PROGRAM PRG_HMI
VAR
	counter	: FB_Counter;
END_VAR

GVL_HMI.output_1:=  GVL_HMI.input_1 AND GVL_HMI.input_2;

counter(CTU:=GVL_HMI.btn_CTU ,
		CTD:=GVL_HMI.btn_CTD , 
		Step:= 1, 
		Value:= GVL_HMI.Counter);

END_PROGRAM

(* stored: Version 1.1.0.1, ProductVersion 3.1.4024.12
   POU PRG_HMI: Id {a018f69f-c419-4915-9b1a-cc5c4ffb9557}, SpecialFunc None *)
